(*

short summary
=============

.. <legal notes>

legal notes
=================
| SPDX-FileCopyrightText: © 2023 ekvip automation GmbH <info@ekvip.de>
| SPDX-License-Identifier: Apache-2.0
| For details check: Apache-2.0_

.. _Apache-2.0: https://www.apache.org/licenses/LICENSE-2.0

.. </legal notes>

*)

INTERFACE IAttachAssertorContainer EXTENDS  __SYSTEM.IQueryInterface

(*

short summary
=============

.. <legal notes>

legal notes
=================
| SPDX-FileCopyrightText: © 2023 ekvip automation GmbH <info@ekvip.de>
| SPDX-License-Identifier: Apache-2.0
| For details check: Apache-2.0_

.. _Apache-2.0: https://www.apache.org/licenses/LICENSE-2.0

.. </legal notes>

*)

PROPERTY attachAssertorContainer : IAssertorContainer
SET
END_SET
END_PROPERTY

END_INTERFACE

(* stored: Version 1.1.0.1, ProductVersion 3.1.4026.12
   Itf IAttachAssertorContainer: Id {fde88d91-cf83-470c-ba30-446634bab73b}
   Property attachAssertorContainer: Id {70ba9d15-9c7b-43e0-9240-ad9c754cbaf4}
   Set Set: Id {6d2871be-447a-4d8e-a07b-e56f5ad7b1d2} *)
